// TIA Portal V17 export
// export: Created 2025-03-07T09:19:47.3056383Z, ExportSetting WithDefaults, DisplayName Totally Integrated Automation Portal, DisplayVersion V17 Update 8, DisplayName TIA Portal Openness, DisplayVersion V17 Update 8, DisplayName TIA Portal Version Control Interface, DisplayVersion V17, DisplayName SINAMICS Startdrive Advanced, DisplayVersion V17 SP2, DisplayName SINAMICS Startdrive G110M, G120, G120C, G120D, G120P, G115D, DisplayVersion V17 SP2, DisplayName SINAMICS Startdrive G130, G150, S120, S150, SINAMICS MV, S210, DisplayVersion V17 SP2, DisplayName STEP 7 Professional, DisplayVersion V17 Update 8, DisplayName SINUMERIK ONE STEP 7 Toolbox, DisplayVersion V17 Update 12, DisplayName SINUMERIK 840D sl STEP 7 Toolbox, DisplayVersion V17 Update 12, DisplayName STEP 7 Safety, DisplayVersion V17 Update 6, DisplayName WinCC Advanced, DisplayVersion V17 Update 8
TYPE "HT10_ENABLE_CHANGE"
// stored: IsFailsafeCompliant false
   STRUCT
      GENERAL_CONDITIONS : Bool;   // GENERAL CONDITIONS
      INTIAL_CONDITIONS : Bool;   // INTIAL CONDITIONS
      MANUAL_REQUEST : Bool;   // MANUAL REQUEST
      GLOBAL_REQUEST : Bool;   // GLOBAL REQUEST
      GLOBAL_REQUEST_RETURN : Bool;   // GLOBAL REQUEST RETURN
      CONTROL_PANEL : Bool;   // CONTROL PANEL
      SELECTED : Bool;   // SELECTED
      HELP : Bool;   // HELP
      PULSE : Bool;   // PULSE
      PULSE_1 : Bool;   // PULSE 1
      PULSE_2 : Bool;   // PULSE 2
      PULSE_3 : Bool;   // PULSE 3
      PULSE_4 : Bool;   // PULSE 4
      GENERAL_CONDITIONS_HELP : Bool;   // GENERAL CONDITIONS HELP
      INITIAL_CONDITIONS_HELP : Bool;   // INITIAL CONDITIONS HELP
   END_STRUCT;
END_TYPE
